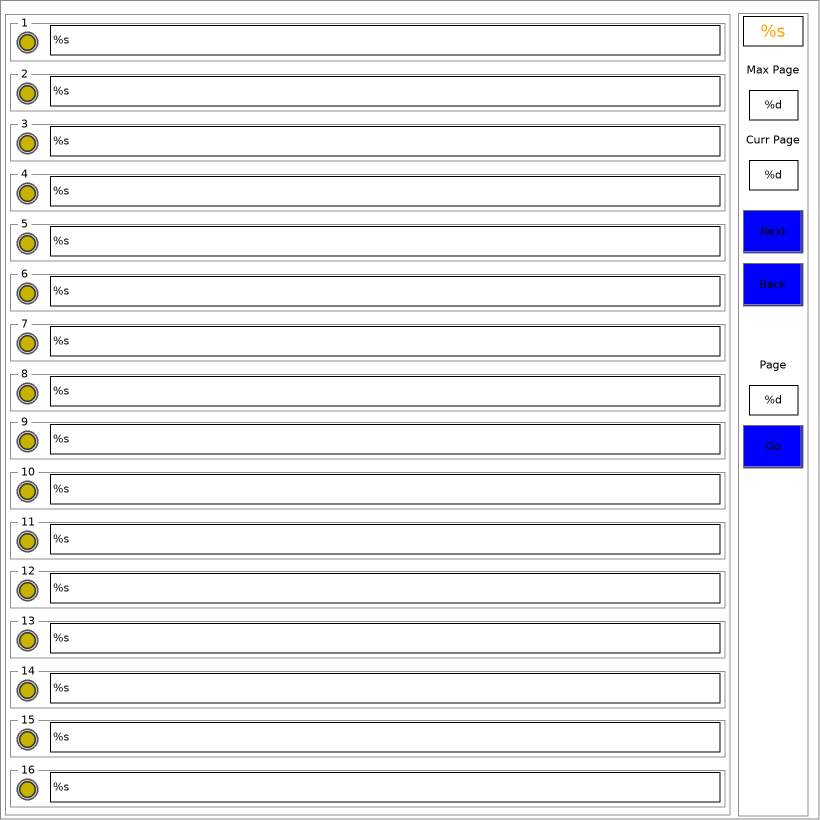
VISUALIZATION IOBase_Show_New  // 820x820
VAR_IN_OUT
	userData:ST_IOBase_Show_HMI;
END_VAR
    GroupBox (5,6 725x809)
        GroupBox (5,9 715x46), "1"
            Lamp1 (5,15 25x25), variable: userData.bIO[1], style: Lamp-Lamp1-Yellow
            Rectangle (40,10 670x30), "%s", text variable: userData.sInfor[1]
        GroupBox (5,60 715x45), "2"
            Lamp1 (5,15 25x25), variable: userData.bIO[2], style: Lamp-Lamp1-Yellow
            Rectangle (40,10 670x30), "%s", text variable: userData.sInfor[2]
        GroupBox (5,110 715x45), "3"
            Lamp1 (5,15 25x25), variable: userData.bIO[3], style: Lamp-Lamp1-Yellow
            Rectangle (40,10 670x30), "%s", text variable: userData.sInfor[3]
        GroupBox (5,160 715x45), "4"
            Lamp1 (5,15 25x25), variable: userData.bIO[4], style: Lamp-Lamp1-Yellow
            Rectangle (40,10 670x30), "%s", text variable: userData.sInfor[4]
        GroupBox (5,210 715x45), "5"
            Lamp1 (5,15 25x25), variable: userData.bIO[5], style: Lamp-Lamp1-Yellow
            Rectangle (40,10 670x30), "%s", text variable: userData.sInfor[5]
        GroupBox (5,260 715x45), "6"
            Lamp1 (5,15 25x25), variable: userData.bIO[6], style: Lamp-Lamp1-Yellow
            Rectangle (40,10 670x30), "%s", text variable: userData.sInfor[6]
        GroupBox (5,310 715x45), "7"
            Lamp1 (5,15 25x25), variable: userData.bIO[7], style: Lamp-Lamp1-Yellow
            Rectangle (40,10 670x30), "%s", text variable: userData.sInfor[7]
        GroupBox (5,360 715x45), "8"
            Lamp1 (5,15 25x25), variable: userData.bIO[8], style: Lamp-Lamp1-Yellow
            Rectangle (40,10 670x30), "%s", text variable: userData.sInfor[8]
        GroupBox (5,408 715x45), "9"
            Lamp1 (5,15 25x25), variable: userData.bIO[9], style: Lamp-Lamp1-Yellow
            Rectangle (40,10 670x30), "%s", text variable: userData.sInfor[9]
        GroupBox (5,458 715x45), "10"
            Lamp1 (5,15 25x25), variable: userData.bIO[10], style: Lamp-Lamp1-Yellow
            Rectangle (40,10 670x30), "%s", text variable: userData.sInfor[10]
        GroupBox (5,508 715x45), "11"
            Lamp1 (5,15 25x25), variable: userData.bIO[11], style: Lamp-Lamp1-Yellow
            Rectangle (40,10 670x30), "%s", text variable: userData.sInfor[11]
        GroupBox (5,557 715x45), "12"
            Lamp1 (5,15 25x25), variable: userData.bIO[12], style: Lamp-Lamp1-Yellow
            Rectangle (40,10 670x30), "%s", text variable: userData.sInfor[12]
        GroupBox (5,607 715x45), "13"
            Lamp1 (5,15 25x25), variable: userData.bIO[13], style: Lamp-Lamp1-Yellow
            Rectangle (40,10 670x30), "%s", text variable: userData.sInfor[13]
        GroupBox (5,657 715x45), "14"
            Lamp1 (5,15 25x25), variable: userData.bIO[14], style: Lamp-Lamp1-Yellow
            Rectangle (40,10 670x30), "%s", text variable: userData.sInfor[14]
        GroupBox (5,706 715x45), "15"
            Lamp1 (5,15 25x25), variable: userData.bIO[15], style: Lamp-Lamp1-Yellow
            Rectangle (40,10 670x30), "%s", text variable: userData.sInfor[15]
        GroupBox (5,756 715x45), "16"
            Lamp1 (5,15 25x25), variable: userData.bIO[16], style: Lamp-Lamp1-Yellow
            Rectangle (40,10 670x30), "%s", text variable: userData.sInfor[16]
    GroupBox (738,5 70x811)
        Button (5,205 60x43), "Next"
            tap userData.bNextPage
        Button (5,258 60x43), "Back"
            tap userData.bBackPage
        Rectangle (11,85 49x30), "%d", text variable: userData.iMaxPage
        Rectangle (11,155 49x30), "%d", text variable: userData.iCurrPage
        Rectangle (11,380 49x30), "%d", text variable: userData.iTargerPage
            OnMouseUp: write the text variable via Default, min 1, max 99
        Button (5,420 60x43), "Go"
            tap userData.bTargerPage
        Label (5,50 60x30), "Max Page"
        Label (5,120 60x30), "Curr Page"
        Label (5,345 60x30), "Page"
        Rectangle (5,11 60x30), "%s", text variable: userData.sIOType
END_VISUALIZATION

(* stored: Version 1.1.0.1, ProductVersion 3.1.4024.4
   Visu IOBase_Show_New: Id {59703ce5-a9db-4c1e-91b4-6463722f6372} *)
